TYPE SAI_Range :
STRUCT
	{attribute addProperty Name "Range"}
	Range AT %Q* : SAI_RangeControl;
END_STRUCT
END_TYPE

(* stored: Version 1.1.0.1, ProductVersion 3.1.4024.9
   DUT SAI_Range: Id {1947960b-e22d-0dfe-005e-1420ae8a6d98} *)
